(* CODESYS project TcpIp.library
   Company: Ziga Javornik
   DefaultNamespace: ZigaLibs.TcpIp
   Version: 0.0.2.2
   Placeholder: ZigaLibs.TcpIp
   Author: Ziga Javornik
   Description: TcpIp communication protocol implementation and various encapsulations of already existing system functions.
   Title: ZigaLibs.TcpIp

Project tree, tasks and I/O mapping:
  libraries: Tc2_Standard, * (Beckhoff Automation GmbH); Tc2_System, * (Beckhoff Automation GmbH); Tc2_TcpIp, * (Beckhoff Automation GmbH); Tc3_Module, * (Beckhoff Automation GmbH); TcUnit, 1.3.1 (www.tcunit.org); ZigaLibs.Core, 0.0.3.7 (Ziga Javornik); ZigaLibs.Logging, 0.0.4.1 (Ziga Javornik)
  GVLs/
  SOURCE/
    TcpIp/
      DUTs/
        data type E_SocketReceiveState
        data type E_SocketSendState
        data type T_Port
      POUs/
        function block FB_TcpIpCommControl [ST]: FB_init, GetLogPrefix, WriteErrorLog, WriteInfoLog, Connect, Disconnect, Receive, Send, Error, IsConnected, ReconnectPeriod
        interface I_TcpIpCommControl: Connect, Disconnect, Error, IsConnected, Receive, ReconnectPeriod, Send
        program TcpIpHelper [ST]: CloseAllSockets
  TESTS/
    Test suites/
      function block FB_TcpIpCommControl_Tests [ST]: Test01_AttemptToConnect_ExpectError
    program PRG_TESTS [ST]
*)

// SOURCE/TcpIp/DUTs/E_SocketReceiveState
{attribute 'qualified_only'}
{attribute 'strict'}
TYPE E_SocketReceiveState :
(
	READY,
	RECEIVING,
	DONE,
	ERROR
);
END_TYPE

// SOURCE/TcpIp/DUTs/E_SocketSendState
{attribute 'qualified_only'}
{attribute 'strict'}
TYPE E_SocketSendState :
(
	READY,
	SENDING,
	DONE,
	ERROR
);
END_TYPE

// SOURCE/TcpIp/DUTs/T_Port
TYPE T_Port : UINT; END_TYPE

// SOURCE/TcpIp/POUs/FB_TcpIpCommControl
// A function block for TcpIp control. Body should be called, 
// but all the logic is done with method calling and awaiting "TRUE" returned when the method finishes.
FUNCTION_BLOCK FB_TcpIpCommControl 
EXTENDS ZigaLibs_Core.FB_HasInstanceNameAndPath 
IMPLEMENTS I_TcpIpCommControl

VAR
	_error					: BOOL;
	_errorReceiving			: BOOL;
	_errorSending			: BOOL;
	_isConnected			: BOOL;
	_clientServerControl	: Tc2_TcpIp.FB_ClientServerConnection;
	_socketHandle			: Tc2_TcpIp.T_HSOCKET;
	_logger					: REFERENCE TO ZigaLibs_Logging.I_Logger;
END_VAR

_clientServerControl(nMode := Tc2_TcpIp.CONNECT_MODE_ENABLEDBG, hSocket => _socketHandle);
_error := _errorReceiving OR _errorSending OR _clientServerControl.bError;

METHOD FB_init : BOOL
VAR_INPUT
	bInitRetains 	: BOOL; // if TRUE, the retain variables are initialized (warm start / cold start)
	bInCopyCode 	: BOOL;  // if TRUE, the instance afterwards gets moved into the copy code (online change)
	logger			: REFERENCE TO ZigaLibs_Logging.I_Logger;
END_VAR
_logger REF= logger;
END_METHOD

METHOD GetLogPrefix : STRING
VAR_INPUT
END_VAR
GetLogPrefix := Tc2_Standard.CONCAT(THIS^.InstancePath, ': ');
END_METHOD

METHOD WriteErrorLog
VAR_INPUT
	message	: Tc2_System.T_MaxString;
END_VAR
IF NOT __ISVALIDREF(_logger) THEN
	RETURN;
END_IF

_logger.LogError(Tc2_Standard.CONCAT(THIS^.GetLogPrefix(), (message)));
END_METHOD

METHOD WriteInfoLog
VAR_INPUT
	message	: Tc2_System.T_MaxString;
END_VAR
IF NOT __ISVALIDREF(_logger) THEN
	RETURN;
END_IF

_logger.LogInfo(Tc2_Standard.CONCAT(THIS^.GetLogPrefix(), (message)));
END_METHOD

// Connets to the target client with the provided Ip address and port
METHOD Connect : BOOL
VAR_INPUT
	Ipv4Address	: Tc2_System.T_IPv4Addr;	// Ip Address
	Port		: UINT;	// Port
END_VAR
VAR_INST
	connected	: R_TRIG;
END_VAR
VAR
	sb	: ZigaLibs_Core.FB_StringBuilder;
END_VAR
connected(CLK := _clientServerControl.eState = Tc2_TcpIp.E_SocketConnectionState.eSOCKET_CONNECTED AND NOT _clientServerControl.bError);

IF connected.Q THEN
	sb.AddString('Connected to')
		.AddWithQuotationMark(_clientServerControl.sRemoteHost)
		.AddString(' with port ')
		.AddAny(_clientServerControl.nRemotePort);
	THIS^.WriteInfoLog(sb.Create());
END_IF

IF THIS^.IsConnected = FALSE THEN
	_clientServerControl.bEnable := TRUE;
	_clientServerControl.sRemoteHost := Ipv4Address;
	_clientServerControl.nRemotePort := Port;
	_clientServerControl.sSrvNetID := '';
ELSE
	Connect := TRUE;
END_IF
END_METHOD

// Disconnects from the server and closes all active socket connections. Returns TRUE when done.
METHOD Disconnect : BOOL
VAR_INST
	disconnected	: Tc2_Standard.F_TRIG;
END_VAR
VAR
	sb			: ZigaLibs_Core.FB_StringBuilder;
END_VAR
disconnected(CLK := THIS^.IsConnected AND NOT THIS^.Error);

IF disconnected.Q THEN
	sb.AddString('Disconnected from ')
		.AddWithQuotationMark(_clientServerControl.sRemoteHost)
		.AddString(' with port ')
		.AddAny(_clientServerControl.nRemotePort);
	THIS^.WriteInfoLog(sb.Create());
END_IF

IF _clientServerControl.bEnable THEN
	_clientServerControl.bEnable := FALSE;
END_IF

_errorSending := FALSE;
_errorReceiving := FALSE;

Disconnect := _clientServerControl.eState = Tc2_TcpIp.E_SocketConnectionState.eSOCKET_DISCONNECTED;
END_METHOD

// Awaits a response from the client and returns TRUE when done. Response string can be found in the refResponse
// Method needs to be called untill TRUE is returned to finish the sending sequence!
METHOD Receive : BOOL
VAR_INPUT
	refResponse	: REFERENCE TO Tc2_System.T_MaxString;	// Response will be written to the string variable here
END_VAR

VAR_INST
	sResponse			: Tc2_System.T_MaxString;
	eSocketReceiveState	: E_SocketReceiveState;
	fbSocketReceive		: Tc2_TcpIp.FB_SocketReceive;
	bReceiveError		: BOOL;
END_VAR
VAR
	sb	: ZigaLibs_Core.FB_StringBuilder;
END_VAR
CASE eSocketReceiveState OF
	E_SocketReceiveState.READY:
		fbSocketReceive(bExecute := FALSE);
		IF THIS^.IsConnected THEN
			bReceiveError := FALSE;
			fbSocketReceive(
				bExecute := TRUE,
				cbLen := SIZEOF(refResponse),
				pDest := ADR(refResponse),
				sSrvNetId := '',
				hSocket := _socketHandle);
			eSocketReceiveState := E_SocketReceiveState.RECEIVING;
		END_IF
	
	E_SocketReceiveState.RECEIVING:
		fbSocketReceive(bExecute := FALSE);
		IF NOT fbSocketReceive.bError AND_THEN NOT fbSocketReceive.bBusy THEN
			eSocketReceiveState := E_SocketReceiveState.DONE;
		ELSIF fbSocketReceive.bError THEN
			eSocketReceiveState := E_SocketReceiveState.ERROR;	
		END_IF
	
	E_SocketReceiveState.DONE:
		Receive := TRUE;
		eSocketReceiveState := E_SocketReceiveState.READY;
	
	E_SocketReceiveState.ERROR:
		bReceiveError := TRUE;
		eSocketReceiveState := E_SocketReceiveState.DONE;
		
		sb.AddString('Error while receiving from ')
			.AddWithDblQuotationMarks(_socketHandle.remoteAddr.sAddr)
			.AddString('. Error code received is ')
			.AddWithQuotationMark(TO_STRING(fbSocketReceive.nErrId));
		THIS^.WriteErrorLog(sb.Create());
END_CASE

_errorReceiving := bReceiveError;
END_METHOD

// Sends the command to the client and returns TRUE when done. 
// Method needs to be called untill TRUE is returned to finish the sending sequence!
METHOD Send : BOOL
VAR_INPUT
	sCommand	: Tc2_System.T_MaxString;	// Command to be send
END_VAR
VAR_INST
	fbSocketSend		: Tc2_TcpIp.FB_SocketSend;
	eSsocketSendState	: E_SocketSendState;
	arrSendDataBytes	: ARRAY[0..255] OF BYTE;
	nSendDataCount		: UDINT;
	bSendError			: BOOL;
END_VAR

VAR
	sb	: ZigaLibs_Core.FB_StringBuilder;
END_VAR
CASE eSsocketSendState OF
	E_SocketSendState.READY:
		bSendError := FALSE;
		IF sCommand <> '' THEN
			// Clear array for new data
			Tc2_System.MEMSET(
				destAddr := ADR(arrSendDataBytes),
				n := SIZEOF(arrSendDataBytes),
				fillByte := 0);
				
			// Prepare data
			Tc2_System.MEMCPY(
				destAddr := ADR(arrSendDataBytes),
				n := SIZEOF(sCommand),
				srcAddr := ADR(sCommand));
				
			// Get the data count, no empty bytes
			nSendDataCount := 0;
			FOR nSendDataCount := 0 TO SIZEOF(arrSendDataBytes) BY 1 DO
				IF arrSendDataBytes[nSendDataCount] = 0 THEN
					EXIT;
				END_IF
			END_FOR

			// Send data
			fbSocketSend(
				bExecute := TRUE,
				cbLen := nSendDataCount,
				pSrc := ADR(arrSendDataBytes),
				hSocket := _socketHandle);
				
			eSsocketSendState := E_SocketSendState.SENDING;
		END_IF
	
	E_SocketSendState.SENDING:
		fbSocketSend(bExecute := FALSE);
		IF fbSocketSend.bError THEN 
			eSsocketSendState := E_SocketSendState.ERROR;
		ELSIF fbSocketSend.bBusy = FALSE THEN
				eSsocketSendState := E_SocketSendState.DONE;
		END_IF
		
	E_SocketSendState.DONE:
		Send := TRUE;
		eSsocketSendState := E_SocketSendState.READY;
		
	E_SocketSendState.ERROR:
		bSendError := TRUE;
		eSsocketSendState := E_SocketSendState.DONE;
		sb.AddString('Error while sending from ')
			.AddWithQuotationMark(_socketHandle.localAddr.sAddr)
			.AddString(' to ')
			.AddWithDblQuotationMarks(_socketHandle.remoteAddr.sAddr)
			.AddString('. Command being sent was ')
			.AddWithQuotationMark(sCommand)
			.AddString('. Error code received is ')
			.AddWithQuotationMark(TO_STRING(fbSocketSend.nErrId));
		THIS^.WriteErrorLog(sb.Create());
		
END_CASE

_errorSending := bSendError;
END_METHOD

{attribute 'monitoring' := 'call'}
PROPERTY Error : BOOL
GET
Error := _error;
END_GET
END_PROPERTY

{attribute 'monitoring' := 'call'}
PROPERTY PUBLIC IsConnected : BOOL
GET
IsConnected := _clientServerControl.eState = Tc2_TcpIp.E_SocketConnectionState.eSOCKET_CONNECTED;
END_GET
END_PROPERTY

{attribute 'monitoring' := 'call'}
(* Gets or sets the reconnect period. 
The value should not be set too low, since timeout periods of > 30 s may occur in the event of a network interruption. 
If the value is too low, command execution would be interrupted prematurely, and ADS error code 1861 (timeout elapsed) 
would be returned instead of the Winsocket error WSAETIMEDOUT.*)
PROPERTY PUBLIC ReconnectPeriod : TIME
GET
ReconnectPeriod := _clientServerControl.tReconnect;
END_GET
SET
IF ReconnectPeriod > T#30S THEN
	_clientServerControl.tReconnect := ReconnectPeriod;
END_IF
END_SET
END_PROPERTY

END_FUNCTION_BLOCK

// SOURCE/TcpIp/POUs/I_TcpIpCommControl
// An interface for a fully functioning TCPIP control with only method calling
INTERFACE I_TcpIpCommControl

// Connets to the target client with the provided Ip address and port
METHOD Connect : BOOL
VAR_INPUT
	Ipv4Address	: Tc2_System.T_IPv4Addr;	// Ip Address
	Port		: UINT;	// Port
END_VAR
END_METHOD

// Disconnects from the server and closes all active socket connections. Returns TRUE when done.
METHOD Disconnect : BOOL
END_METHOD

{attribute 'monitoring' := 'call'}
PROPERTY Error : BOOL
GET
END_GET
END_PROPERTY

{attribute 'monitoring' := 'call'}
PROPERTY PUBLIC IsConnected : BOOL
GET
END_GET
END_PROPERTY

// Awaits a response from the client and returns TRUE when done. Response string can be found in the refResponse
// Method needs to be called untill TRUE is returned to finish the sending sequence!
METHOD Receive : BOOL
VAR_INPUT
	refResponse	: REFERENCE TO Tc2_System.T_MaxString;	// Response will be written to the string variable here
END_VAR
END_METHOD

{attribute 'monitoring' := 'call'}
(* Gets or sets the reconnect period. 
The value should not be set too low, since timeout periods of > 30 s may occur in the event of a network interruption. 
If the value is too low, command execution would be interrupted prematurely, and ADS error code 1861 (timeout elapsed) 
would be returned instead of the Winsocket error WSAETIMEDOUT.*)
PROPERTY PUBLIC ReconnectPeriod : TIME
GET
END_GET
SET
END_SET
END_PROPERTY

// Sends the command to the client and returns TRUE when done. 
// Method needs to be called untill TRUE is returned to finish the sending sequence!
METHOD Send : BOOL
VAR_INPUT
	sCommand	: Tc2_System.T_MaxString;	// Command to be send
END_VAR
END_METHOD

END_INTERFACE

// SOURCE/TcpIp/POUs/TcpIpHelper
// TcpIp helper class
{attribute 'no_explicit_call' := 'Body contains no logic, calling methods only allowed.'}
{attribute 'hide_all_locals'}
PROGRAM TcpIpHelper
VAR
	_socketCloseAll	: Tc2_TcpIp.FB_SocketCloseAll;
	_closeAllState	: (CLOSE_ALL_READY, CLOSE_ALL_BUSY, CLOSE_ALL_DONE);
END_VAR

// Closes all connections on the server that were opened by the PLC runtime system.
// In each PLC runtime system that uses the socket function blocks, an instance of FB_SocketCloseAll should be called during the PLC start.
// Method returns TRUE when done. If an error has ocured it is provided in the outputs.
METHOD PUBLIC CloseAllSockets : BOOL
VAR_INPUT
	serverNetId	: Tc2_System.T_AmsNetID;	// TcpIp server's netID. For local set to empty string
END_VAR
VAR_OUTPUT
	error	: BOOL;		// If an error occurs, the flag will be set to true.
	errorId	: UDINT;	// ErrorId which has ocured when the function calling has finished
END_VAR
_socketCloseAll(sSrvNetId := serverNetId);
CASE _closeAllState OF
	CLOSE_ALL_READY:
		error := FALSE;
		errorId := 0;
		_socketCloseAll.bExecute := TRUE;
		_closeAllState := CLOSE_ALL_BUSY;
		
	CLOSE_ALL_BUSY:
		IF _socketCloseAll.bError  OR NOT _socketcloseAll.bBusy THEN
			_closeAllState := CLOSE_ALL_DONE;
		END_IF
	
	CLOSE_ALL_DONE:
		error := _socketCloseAll.bError;
		errorId := _socketCloseAll.nErrId;
		_socketCloseAll(bExecute := FALSE, sSrvNetId := '');
		CloseAllSockets := TRUE;
END_CASE
END_METHOD

END_PROGRAM

// TESTS/Test suites/FB_TcpIpCommControl_Tests
// Subject under test
FUNCTION_BLOCK INTERNAL FB_TcpIpCommControl_Tests EXTENDS FB_TestSuite

// Create instance variables that will be accesible for all tests
VAR
	_tcpIp	: FB_TcpIpCommControl(0);
END_VAR

// Call your test methods here
_tcpIp();
// Need to realize this with a TCP server... For now disabled
//THIS^.Test01_AttemptToConnect_ExpectError();

METHOD PRIVATE Test01_AttemptToConnect_ExpectError

(* Instanced variables are VERY useful for writing tests since tests are run in paralel (by default).
By instantiating local variables that are not placed on the same stack as method (values are retained between calls)
you make sure that the SUT is not changed by some other test. *)
VAR_INST
	testAddress	: Tc2_System.T_IPv4Addr := '192.168.0.1';
	maxDelayForError	: Tc2_Standard.TON := (PT := T#35S);
END_VAR

// Place temporary variables here
VAR
	
END_VAR
// The name of the test, is the same as method name!
IF TcUnit.TEST_ORDERED('Test01_AttemptToConnect_ExpectError') THEN
	_tcpIp.ReconnectPeriod := T#30S;
	_tcpIp.Connect(Ipv4Address := testAddress, Port := 3232);

	maxDelayForError(IN := TRUE);

	IF maxDelayForError.Q THEN
		AssertTrue(Condition := _tcpIp.Error, Message := '10 seconds after connecting to a non existing address and port, the error should be raised!');
		AssertFalse(Condition := _tcpIp.IsConnected, Message := 'Connecting to a non existing address and port, the IsConnected property should be false!');
		TcUnit.TEST_FINISHED();	
	END_IF
END_IF
END_METHOD

END_FUNCTION_BLOCK

// TESTS/PRG_TESTS
PROGRAM INTERNAL PRG_TESTS

(* Instantiate test suites here. Naming convention for tests should be a suffix with _Tests.
Good practice for creating test methods is to end them with _test as well. *)
VAR
	TcpIpCommControlTests	: FB_TcpIpCommControl_Tests;

END_VAR


// Run tests in paralel
//TcUnit.RUN();

// Run tests in sequence, one after the other. Uncomment if required.
TcUnit.RUN_IN_SEQUENCE();

END_PROGRAM
